(* Logix 5000 project; controller AMANA_DC_PLANT_01 vendor 1 type 14 code 164 rev 31.12; software revision 31.02; part 5 of 9 *)
(* tags used below, declared in another part *)
   Break_1stStation : BOOL;
   LN00_to_DC1_Main_Messages_5 : DINT[120];
   LN00_to_DC1_Main_Messages_6 : DINT[120];
   LN00DEM06 : DINT;
   LN00DEM07 : DINT;
   LN00DEM08 : DINT;
   LN00DEM09 : DINT;
   LN00DEM10 : DINT;
   LN00DEM11 : DINT;
   LN00DEM12 : DINT;
   LN00DEM13 : DINT;
   LN00DEM14 : DINT;
   LN00DEM15 : DINT;
   LN00DEM16 : DINT;
   LN00DEM17 : DINT;
   LN00DEM18 : DINT;
   LN00DEM19 : DINT;
   LN00DEM20 : DINT;
   LN00DEM21 : DINT;
   LN00DEM22 : DINT;
   LN00DEM23 : DINT;
   LN00DEM24 : DINT;
   LN00DEM25 : DINT;
   LN00DEM26 : DINT;
   LN00DEM27 : DINT;
   LN00DEM28 : DINT;
   LN00DEM29 : DINT;
   LN00DEM30 : DINT;
   LN00DEM31 : DINT;
   LN00DEM32 : DINT;
   LN00DEM33 : DINT;
   LN00DEM34 : DINT;
   LN00DEM35 : DINT;
   LN00DEM36 : DINT;
   LN00DEM37 : DINT;
   LN00DEM38 : DINT;
   LN00DEM39 : DINT;
   LN00DEM40 : DINT;
   LN00DEM41 : DINT;
   LN00DEM42 : DINT;
   LN00DEM43 : DINT;
   LN00DEM44 : DINT;
   LN00DEM45 : DINT;
   LN00DEM46 : DINT;
   LN00DEM47 : DINT;
   LN00DEM48 : DINT;
   LN00DEM49 : DINT;
   LN00DEM50 : DINT;
   LN00DEM51 : DINT;
   LN00DEM52 : DINT;
   LN00DEM53 : DINT;
   LN00DEM54 : DINT;
   LN00DEM55 : DINT;
   LN00DEM56 : DINT;
   LN00DEM57 : DINT;
   LN00DEM58 : DINT;
   LN00DEM59 : DINT;
   LN00DEM60 : DINT;
   LN00DEM61 : DINT;
   LN00DEM62 : DINT;
   LN00DEM63 : DINT;
   LN00DEM64 : DINT;
   LN00DEM65 : DINT;
   LN00DEM66 : DINT;
   LN00DEM67 : DINT;
   LN00DEM68 : DINT;
   LN00DEM69 : DINT;
   LN00DEM70 : DINT;
   LN00DEM71 : DINT;
   LN00DEM72 : DINT;
   LN00DEM73 : DINT;
   LN00DEM74 : DINT;
   LN00DEM75 : DINT;
   LN00DEM76 : DINT;
   LN00DEM77 : DINT;
   LN00DEM78 : DINT;
   LN00DEM79 : DINT;
   LN00DEM80 : DINT;
   LN00DEM81 : DINT;
   LN00DEM82 : DINT;
   LN00DEM83 : DINT;
   LN00DEM84 : DINT;
   LN00DEM85 : DINT;
   LN00DEM86 : DINT;
   LN00DEM87 : DINT;
   LN00DEM88 : DINT;
   LN00DEM89 : DINT;
   LN00DEM90 : DINT;
   LN00DEM91 : DINT;
   LN00DEM92 : DINT;
   LN00DEM93 : DINT;
   LN00DEM94 : DINT;
   LN00DEM95 : DINT;
   LN00DEM96 : DINT;
   LN00DEM97 : DINT;
   LN00DEM98 : DINT;
   LN00DFM01 : DINT;
   LN00DFM02 : DINT;
   LN00DFM03 : DINT;
(* LN00, continued *)

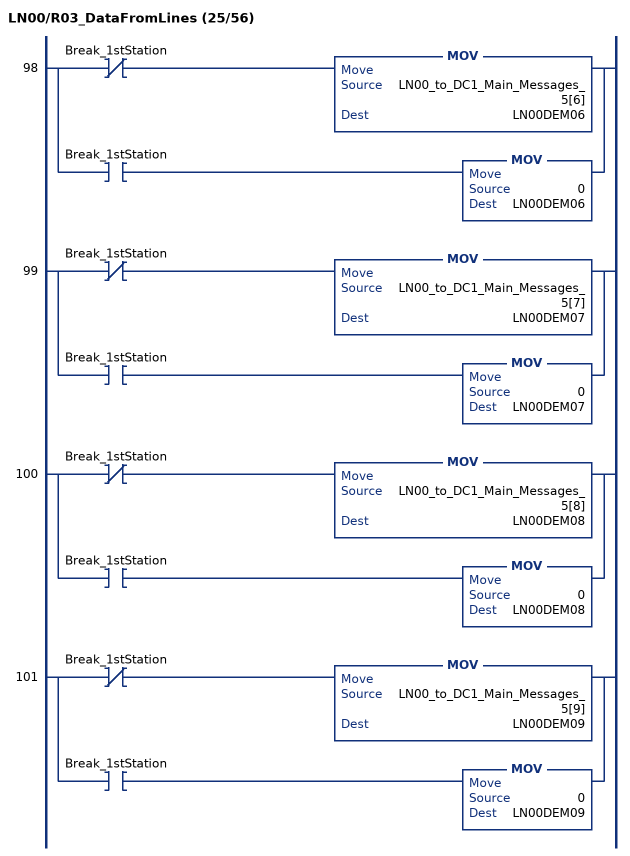
   [picture p71: LN00/R03_DataFromLines rungs 98-101]
   98: [XIO(Break_1stStation) MOV(LN00_to_DC1_Main_Messages_5[6],LN00DEM06) ,XIC(Break_1stStation) MOV(0,LN00DEM06) ];
   99: [XIO(Break_1stStation) MOV(LN00_to_DC1_Main_Messages_5[7],LN00DEM07) ,XIC(Break_1stStation) MOV(0,LN00DEM07) ];
   100: [XIO(Break_1stStation) MOV(LN00_to_DC1_Main_Messages_5[8],LN00DEM08) ,XIC(Break_1stStation) MOV(0,LN00DEM08) ];
   101: [XIO(Break_1stStation) MOV(LN00_to_DC1_Main_Messages_5[9],LN00DEM09) ,XIC(Break_1stStation) MOV(0,LN00DEM09) ];
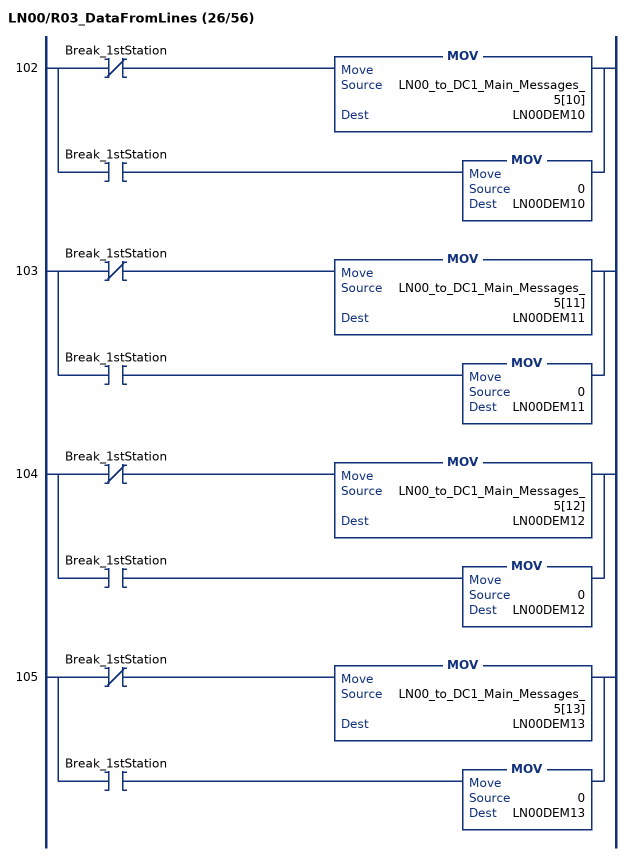
   102: [XIO(Break_1stStation) MOV(LN00_to_DC1_Main_Messages_5[10],LN00DEM10) ,XIC(Break_1stStation) MOV(0,LN00DEM10) ];
   103: [XIO(Break_1stStation) MOV(LN00_to_DC1_Main_Messages_5[11],LN00DEM11) ,XIC(Break_1stStation) MOV(0,LN00DEM11) ];
   104: [XIO(Break_1stStation) MOV(LN00_to_DC1_Main_Messages_5[12],LN00DEM12) ,XIC(Break_1stStation) MOV(0,LN00DEM12) ];
   105: [XIO(Break_1stStation) MOV(LN00_to_DC1_Main_Messages_5[13],LN00DEM13) ,XIC(Break_1stStation) MOV(0,LN00DEM13) ];
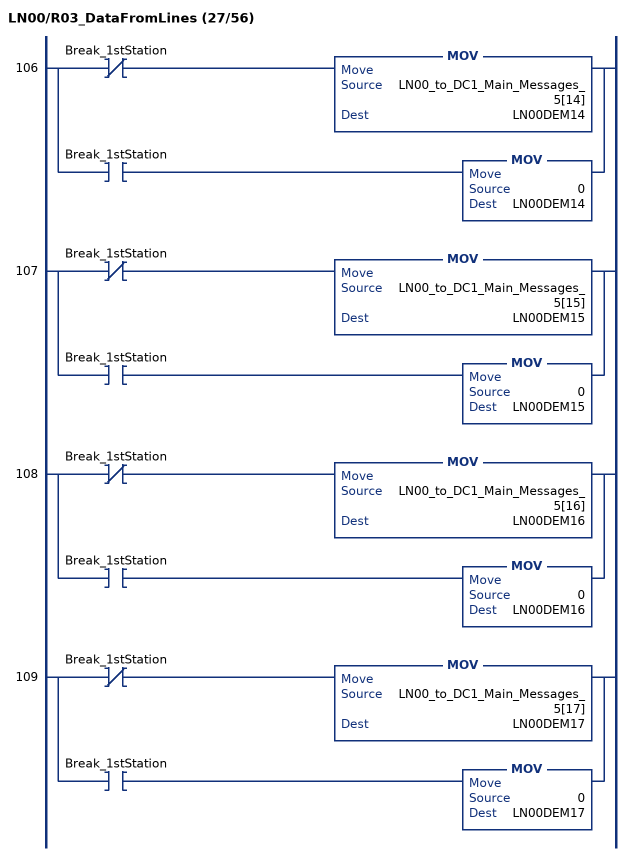
   106: [XIO(Break_1stStation) MOV(LN00_to_DC1_Main_Messages_5[14],LN00DEM14) ,XIC(Break_1stStation) MOV(0,LN00DEM14) ];
   107: [XIO(Break_1stStation) MOV(LN00_to_DC1_Main_Messages_5[15],LN00DEM15) ,XIC(Break_1stStation) MOV(0,LN00DEM15) ];
   108: [XIO(Break_1stStation) MOV(LN00_to_DC1_Main_Messages_5[16],LN00DEM16) ,XIC(Break_1stStation) MOV(0,LN00DEM16) ];
   109: [XIO(Break_1stStation) MOV(LN00_to_DC1_Main_Messages_5[17],LN00DEM17) ,XIC(Break_1stStation) MOV(0,LN00DEM17) ];
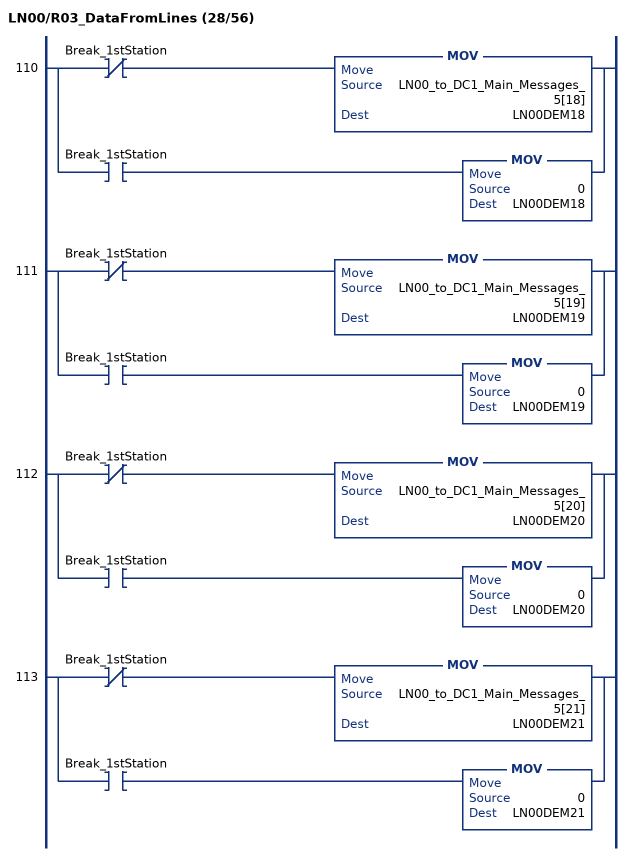
   110: [XIO(Break_1stStation) MOV(LN00_to_DC1_Main_Messages_5[18],LN00DEM18) ,XIC(Break_1stStation) MOV(0,LN00DEM18) ];
   111: [XIO(Break_1stStation) MOV(LN00_to_DC1_Main_Messages_5[19],LN00DEM19) ,XIC(Break_1stStation) MOV(0,LN00DEM19) ];
   112: [XIO(Break_1stStation) MOV(LN00_to_DC1_Main_Messages_5[20],LN00DEM20) ,XIC(Break_1stStation) MOV(0,LN00DEM20) ];
   113: [XIO(Break_1stStation) MOV(LN00_to_DC1_Main_Messages_5[21],LN00DEM21) ,XIC(Break_1stStation) MOV(0,LN00DEM21) ];
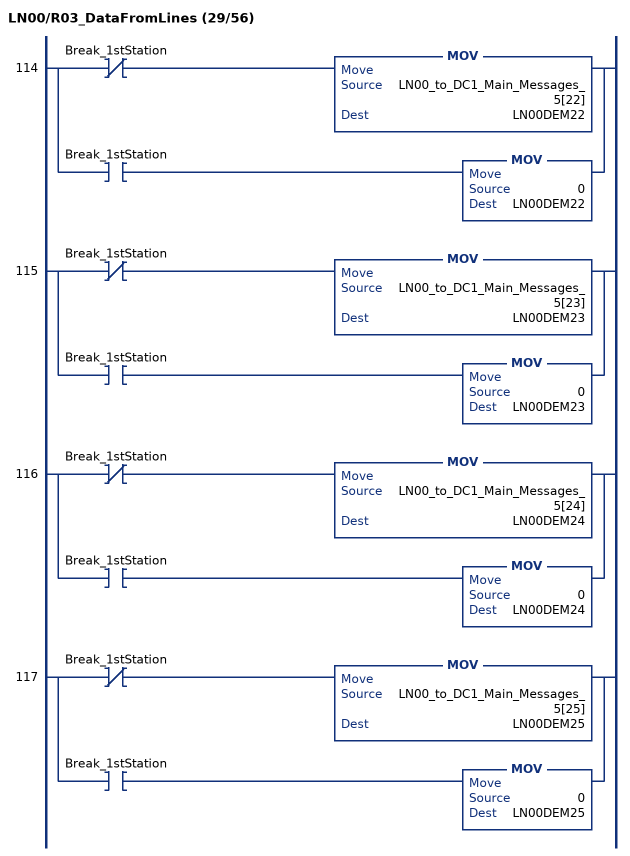
   114: [XIO(Break_1stStation) MOV(LN00_to_DC1_Main_Messages_5[22],LN00DEM22) ,XIC(Break_1stStation) MOV(0,LN00DEM22) ];
   115: [XIO(Break_1stStation) MOV(LN00_to_DC1_Main_Messages_5[23],LN00DEM23) ,XIC(Break_1stStation) MOV(0,LN00DEM23) ];
   116: [XIO(Break_1stStation) MOV(LN00_to_DC1_Main_Messages_5[24],LN00DEM24) ,XIC(Break_1stStation) MOV(0,LN00DEM24) ];
   117: [XIO(Break_1stStation) MOV(LN00_to_DC1_Main_Messages_5[25],LN00DEM25) ,XIC(Break_1stStation) MOV(0,LN00DEM25) ];
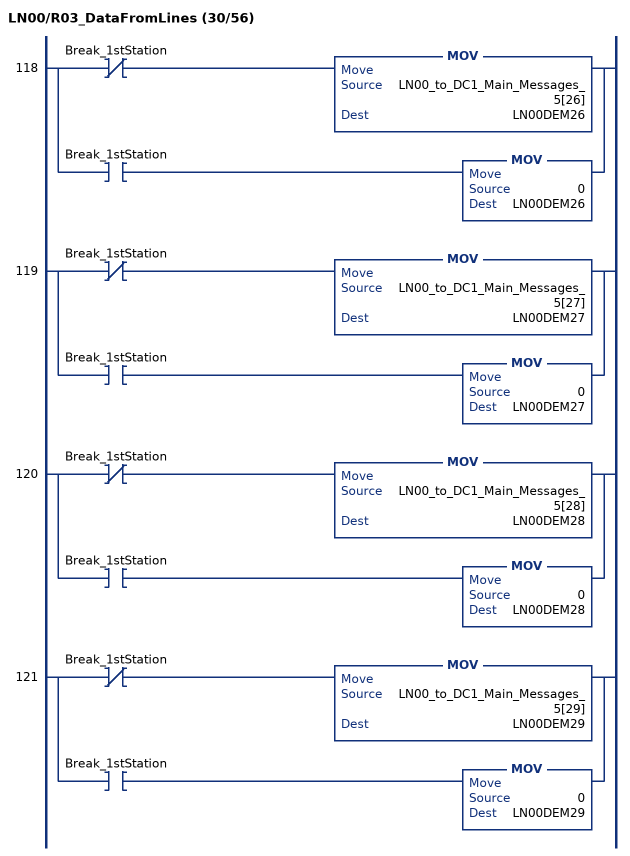
   118: [XIO(Break_1stStation) MOV(LN00_to_DC1_Main_Messages_5[26],LN00DEM26) ,XIC(Break_1stStation) MOV(0,LN00DEM26) ];
   119: [XIO(Break_1stStation) MOV(LN00_to_DC1_Main_Messages_5[27],LN00DEM27) ,XIC(Break_1stStation) MOV(0,LN00DEM27) ];
   120: [XIO(Break_1stStation) MOV(LN00_to_DC1_Main_Messages_5[28],LN00DEM28) ,XIC(Break_1stStation) MOV(0,LN00DEM28) ];
   121: [XIO(Break_1stStation) MOV(LN00_to_DC1_Main_Messages_5[29],LN00DEM29) ,XIC(Break_1stStation) MOV(0,LN00DEM29) ];
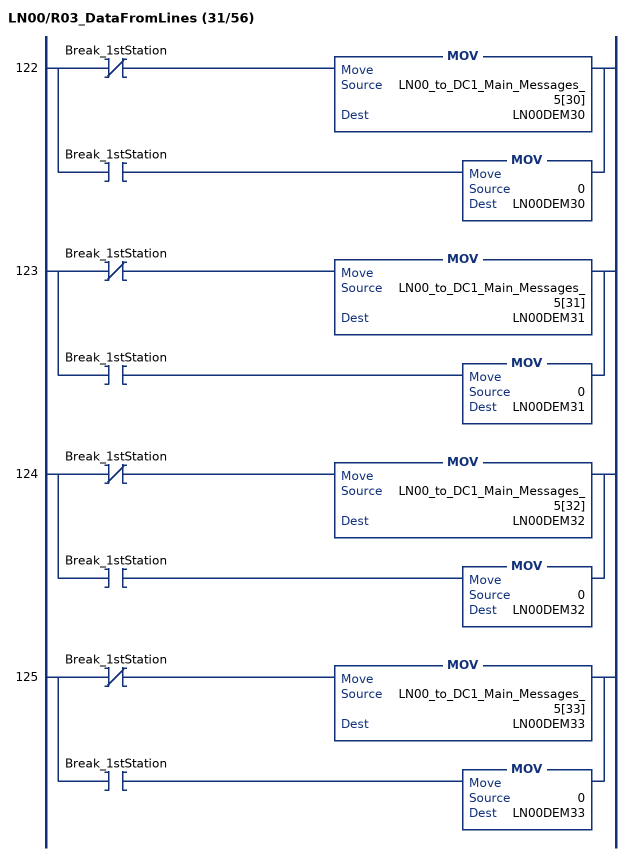
   122: [XIO(Break_1stStation) MOV(LN00_to_DC1_Main_Messages_5[30],LN00DEM30) ,XIC(Break_1stStation) MOV(0,LN00DEM30) ];
   123: [XIO(Break_1stStation) MOV(LN00_to_DC1_Main_Messages_5[31],LN00DEM31) ,XIC(Break_1stStation) MOV(0,LN00DEM31) ];
   124: [XIO(Break_1stStation) MOV(LN00_to_DC1_Main_Messages_5[32],LN00DEM32) ,XIC(Break_1stStation) MOV(0,LN00DEM32) ];
   125: [XIO(Break_1stStation) MOV(LN00_to_DC1_Main_Messages_5[33],LN00DEM33) ,XIC(Break_1stStation) MOV(0,LN00DEM33) ];
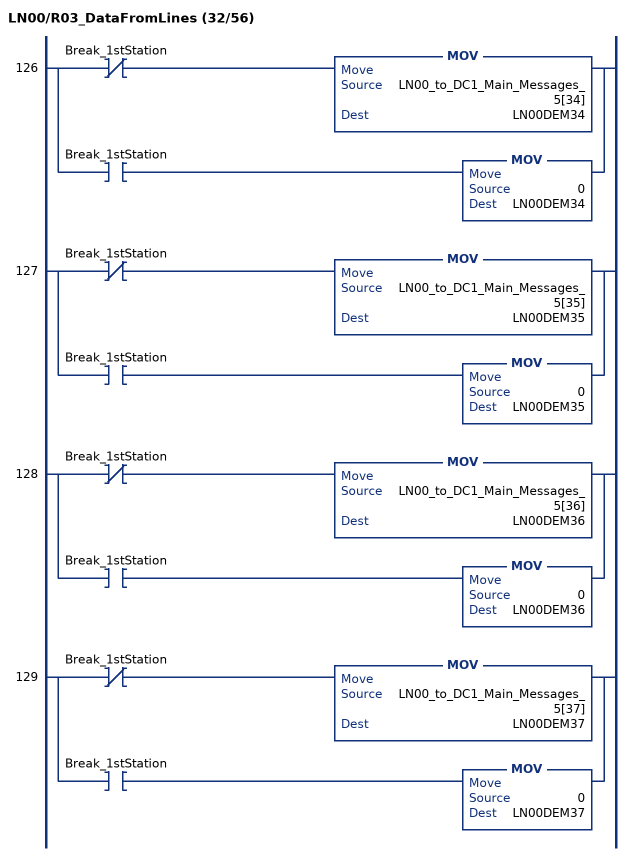
   126: [XIO(Break_1stStation) MOV(LN00_to_DC1_Main_Messages_5[34],LN00DEM34) ,XIC(Break_1stStation) MOV(0,LN00DEM34) ];
   127: [XIO(Break_1stStation) MOV(LN00_to_DC1_Main_Messages_5[35],LN00DEM35) ,XIC(Break_1stStation) MOV(0,LN00DEM35) ];
   128: [XIO(Break_1stStation) MOV(LN00_to_DC1_Main_Messages_5[36],LN00DEM36) ,XIC(Break_1stStation) MOV(0,LN00DEM36) ];
   129: [XIO(Break_1stStation) MOV(LN00_to_DC1_Main_Messages_5[37],LN00DEM37) ,XIC(Break_1stStation) MOV(0,LN00DEM37) ];
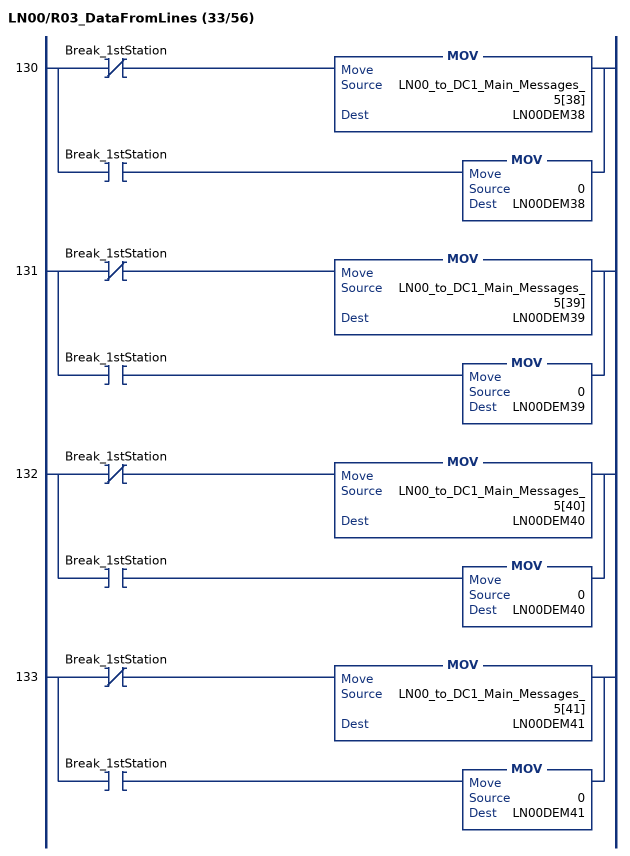
   130: [XIO(Break_1stStation) MOV(LN00_to_DC1_Main_Messages_5[38],LN00DEM38) ,XIC(Break_1stStation) MOV(0,LN00DEM38) ];
   131: [XIO(Break_1stStation) MOV(LN00_to_DC1_Main_Messages_5[39],LN00DEM39) ,XIC(Break_1stStation) MOV(0,LN00DEM39) ];
   132: [XIO(Break_1stStation) MOV(LN00_to_DC1_Main_Messages_5[40],LN00DEM40) ,XIC(Break_1stStation) MOV(0,LN00DEM40) ];
   133: [XIO(Break_1stStation) MOV(LN00_to_DC1_Main_Messages_5[41],LN00DEM41) ,XIC(Break_1stStation) MOV(0,LN00DEM41) ];
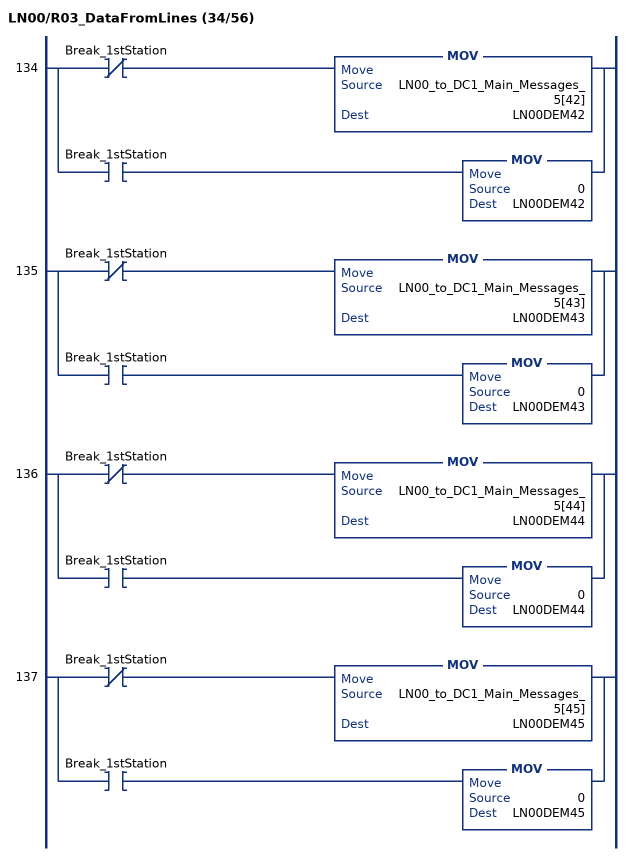
   134: [XIO(Break_1stStation) MOV(LN00_to_DC1_Main_Messages_5[42],LN00DEM42) ,XIC(Break_1stStation) MOV(0,LN00DEM42) ];
   135: [XIO(Break_1stStation) MOV(LN00_to_DC1_Main_Messages_5[43],LN00DEM43) ,XIC(Break_1stStation) MOV(0,LN00DEM43) ];
   136: [XIO(Break_1stStation) MOV(LN00_to_DC1_Main_Messages_5[44],LN00DEM44) ,XIC(Break_1stStation) MOV(0,LN00DEM44) ];
   137: [XIO(Break_1stStation) MOV(LN00_to_DC1_Main_Messages_5[45],LN00DEM45) ,XIC(Break_1stStation) MOV(0,LN00DEM45) ];
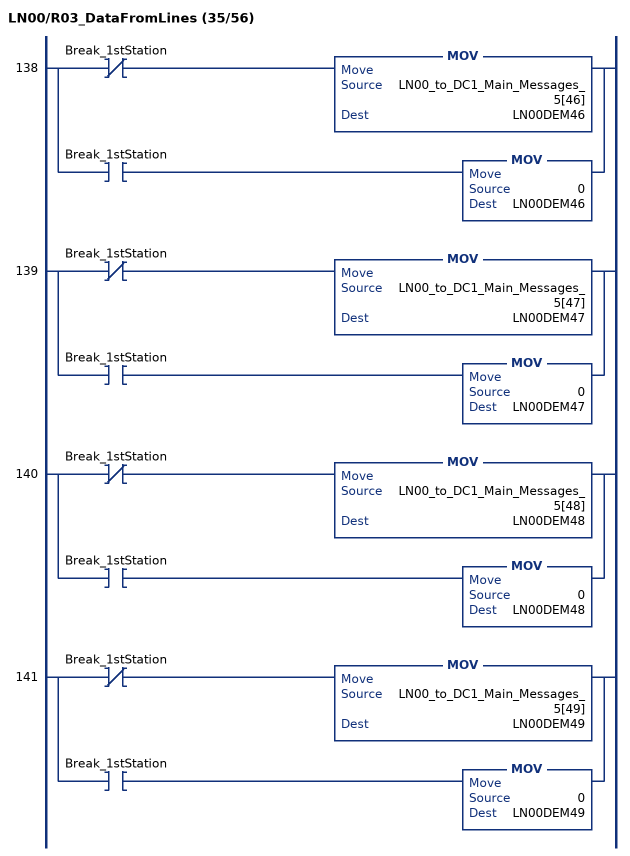
   138: [XIO(Break_1stStation) MOV(LN00_to_DC1_Main_Messages_5[46],LN00DEM46) ,XIC(Break_1stStation) MOV(0,LN00DEM46) ];
   139: [XIO(Break_1stStation) MOV(LN00_to_DC1_Main_Messages_5[47],LN00DEM47) ,XIC(Break_1stStation) MOV(0,LN00DEM47) ];
   140: [XIO(Break_1stStation) MOV(LN00_to_DC1_Main_Messages_5[48],LN00DEM48) ,XIC(Break_1stStation) MOV(0,LN00DEM48) ];
   141: [XIO(Break_1stStation) MOV(LN00_to_DC1_Main_Messages_5[49],LN00DEM49) ,XIC(Break_1stStation) MOV(0,LN00DEM49) ];
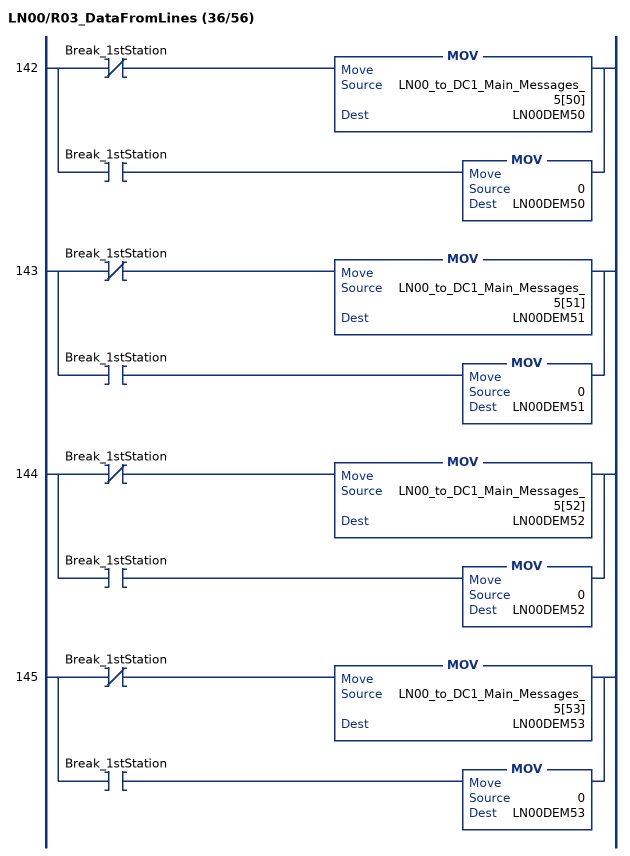
   142: [XIO(Break_1stStation) MOV(LN00_to_DC1_Main_Messages_5[50],LN00DEM50) ,XIC(Break_1stStation) MOV(0,LN00DEM50) ];
   143: [XIO(Break_1stStation) MOV(LN00_to_DC1_Main_Messages_5[51],LN00DEM51) ,XIC(Break_1stStation) MOV(0,LN00DEM51) ];
   144: [XIO(Break_1stStation) MOV(LN00_to_DC1_Main_Messages_5[52],LN00DEM52) ,XIC(Break_1stStation) MOV(0,LN00DEM52) ];
   145: [XIO(Break_1stStation) MOV(LN00_to_DC1_Main_Messages_5[53],LN00DEM53) ,XIC(Break_1stStation) MOV(0,LN00DEM53) ];
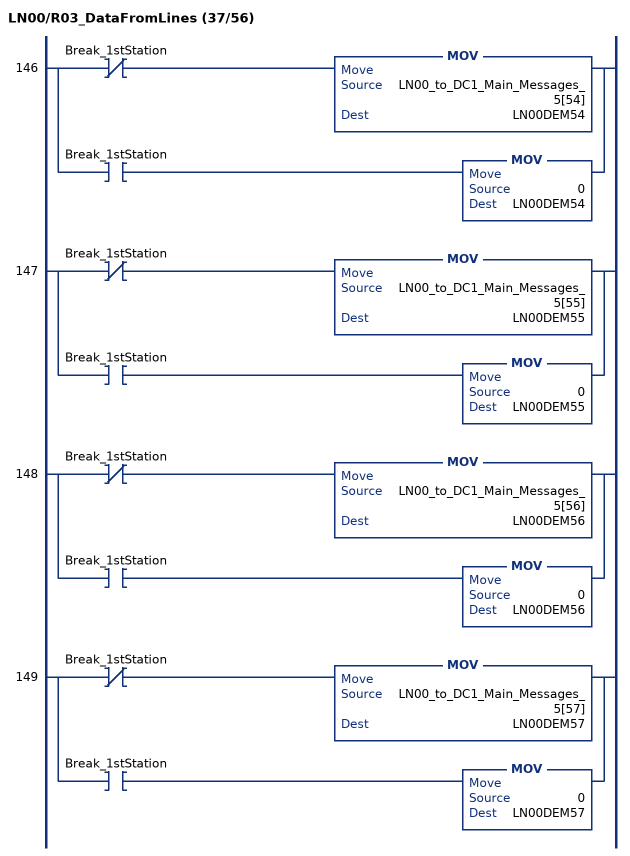
   146: [XIO(Break_1stStation) MOV(LN00_to_DC1_Main_Messages_5[54],LN00DEM54) ,XIC(Break_1stStation) MOV(0,LN00DEM54) ];
   147: [XIO(Break_1stStation) MOV(LN00_to_DC1_Main_Messages_5[55],LN00DEM55) ,XIC(Break_1stStation) MOV(0,LN00DEM55) ];
   148: [XIO(Break_1stStation) MOV(LN00_to_DC1_Main_Messages_5[56],LN00DEM56) ,XIC(Break_1stStation) MOV(0,LN00DEM56) ];
   149: [XIO(Break_1stStation) MOV(LN00_to_DC1_Main_Messages_5[57],LN00DEM57) ,XIC(Break_1stStation) MOV(0,LN00DEM57) ];
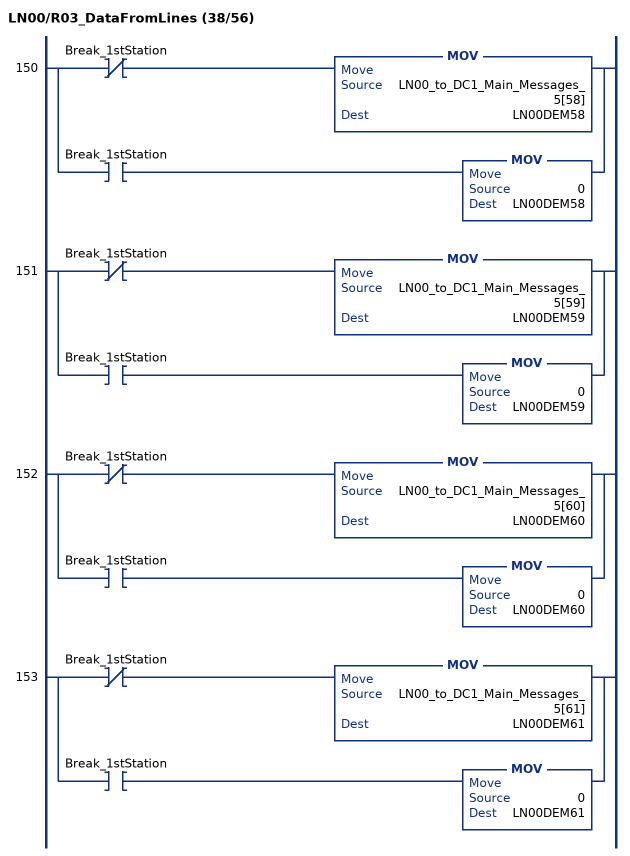
   150: [XIO(Break_1stStation) MOV(LN00_to_DC1_Main_Messages_5[58],LN00DEM58) ,XIC(Break_1stStation) MOV(0,LN00DEM58) ];
   151: [XIO(Break_1stStation) MOV(LN00_to_DC1_Main_Messages_5[59],LN00DEM59) ,XIC(Break_1stStation) MOV(0,LN00DEM59) ];
   152: [XIO(Break_1stStation) MOV(LN00_to_DC1_Main_Messages_5[60],LN00DEM60) ,XIC(Break_1stStation) MOV(0,LN00DEM60) ];
   153: [XIO(Break_1stStation) MOV(LN00_to_DC1_Main_Messages_5[61],LN00DEM61) ,XIC(Break_1stStation) MOV(0,LN00DEM61) ];
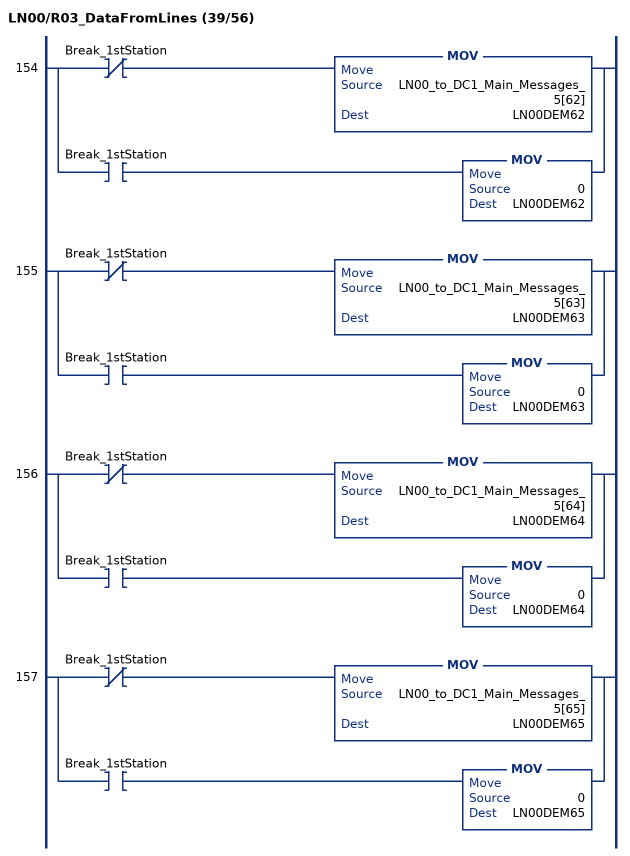
   154: [XIO(Break_1stStation) MOV(LN00_to_DC1_Main_Messages_5[62],LN00DEM62) ,XIC(Break_1stStation) MOV(0,LN00DEM62) ];
   155: [XIO(Break_1stStation) MOV(LN00_to_DC1_Main_Messages_5[63],LN00DEM63) ,XIC(Break_1stStation) MOV(0,LN00DEM63) ];
   156: [XIO(Break_1stStation) MOV(LN00_to_DC1_Main_Messages_5[64],LN00DEM64) ,XIC(Break_1stStation) MOV(0,LN00DEM64) ];
   157: [XIO(Break_1stStation) MOV(LN00_to_DC1_Main_Messages_5[65],LN00DEM65) ,XIC(Break_1stStation) MOV(0,LN00DEM65) ];
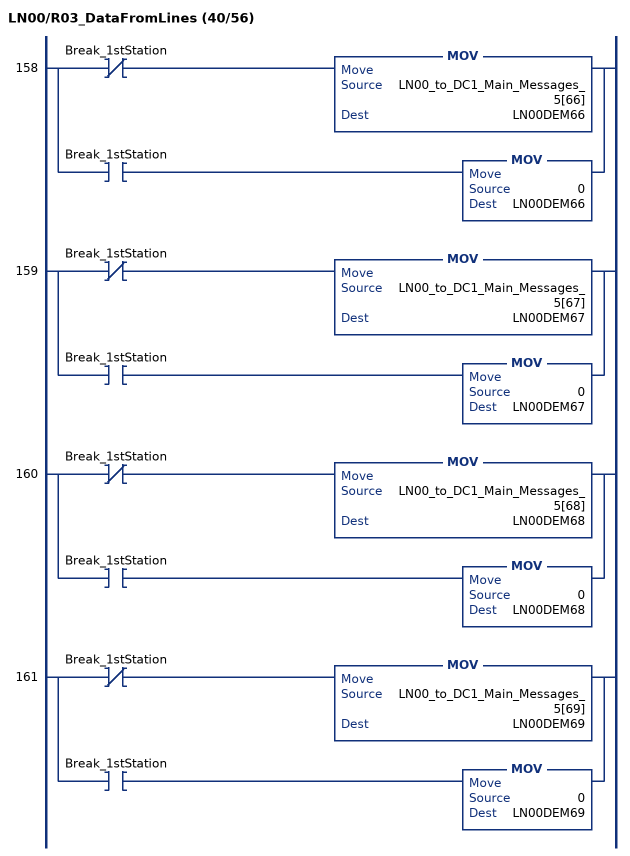
   158: [XIO(Break_1stStation) MOV(LN00_to_DC1_Main_Messages_5[66],LN00DEM66) ,XIC(Break_1stStation) MOV(0,LN00DEM66) ];
   159: [XIO(Break_1stStation) MOV(LN00_to_DC1_Main_Messages_5[67],LN00DEM67) ,XIC(Break_1stStation) MOV(0,LN00DEM67) ];
   160: [XIO(Break_1stStation) MOV(LN00_to_DC1_Main_Messages_5[68],LN00DEM68) ,XIC(Break_1stStation) MOV(0,LN00DEM68) ];
   161: [XIO(Break_1stStation) MOV(LN00_to_DC1_Main_Messages_5[69],LN00DEM69) ,XIC(Break_1stStation) MOV(0,LN00DEM69) ];
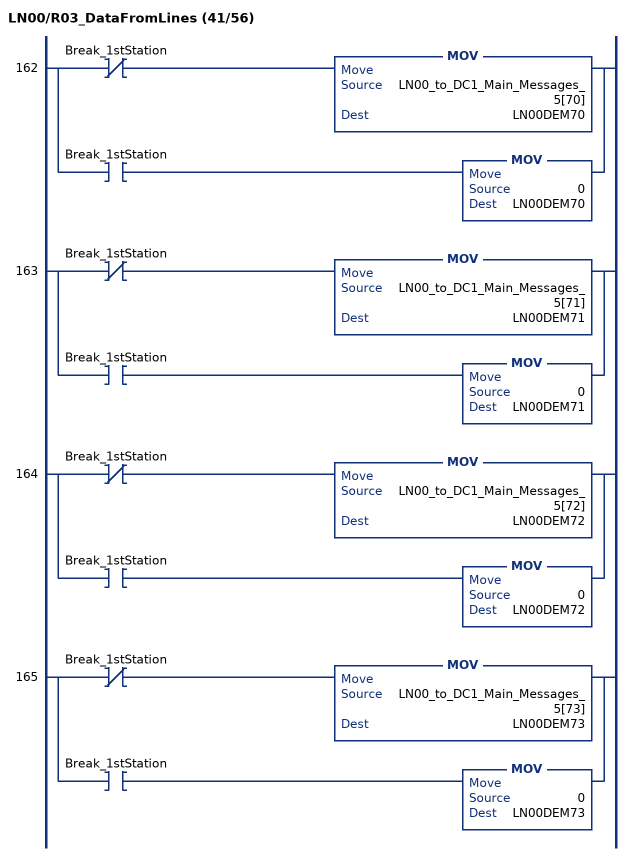
   162: [XIO(Break_1stStation) MOV(LN00_to_DC1_Main_Messages_5[70],LN00DEM70) ,XIC(Break_1stStation) MOV(0,LN00DEM70) ];
   163: [XIO(Break_1stStation) MOV(LN00_to_DC1_Main_Messages_5[71],LN00DEM71) ,XIC(Break_1stStation) MOV(0,LN00DEM71) ];
   164: [XIO(Break_1stStation) MOV(LN00_to_DC1_Main_Messages_5[72],LN00DEM72) ,XIC(Break_1stStation) MOV(0,LN00DEM72) ];
   165: [XIO(Break_1stStation) MOV(LN00_to_DC1_Main_Messages_5[73],LN00DEM73) ,XIC(Break_1stStation) MOV(0,LN00DEM73) ];
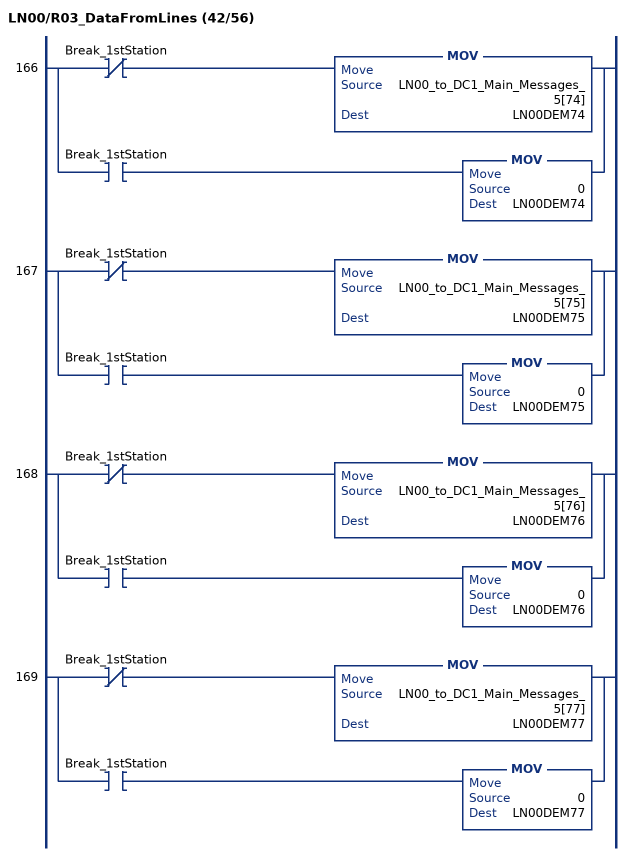
   166: [XIO(Break_1stStation) MOV(LN00_to_DC1_Main_Messages_5[74],LN00DEM74) ,XIC(Break_1stStation) MOV(0,LN00DEM74) ];
   167: [XIO(Break_1stStation) MOV(LN00_to_DC1_Main_Messages_5[75],LN00DEM75) ,XIC(Break_1stStation) MOV(0,LN00DEM75) ];
   168: [XIO(Break_1stStation) MOV(LN00_to_DC1_Main_Messages_5[76],LN00DEM76) ,XIC(Break_1stStation) MOV(0,LN00DEM76) ];
   169: [XIO(Break_1stStation) MOV(LN00_to_DC1_Main_Messages_5[77],LN00DEM77) ,XIC(Break_1stStation) MOV(0,LN00DEM77) ];
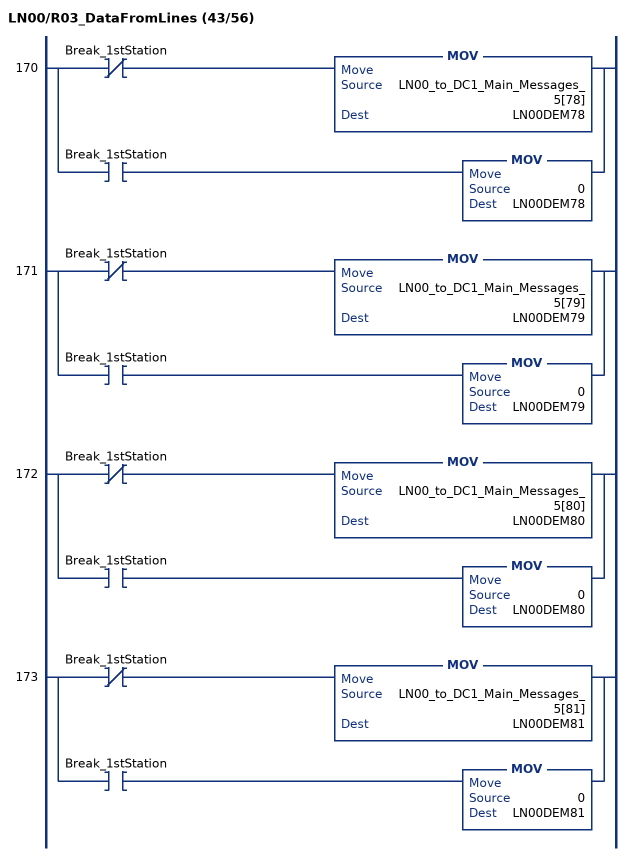
   170: [XIO(Break_1stStation) MOV(LN00_to_DC1_Main_Messages_5[78],LN00DEM78) ,XIC(Break_1stStation) MOV(0,LN00DEM78) ];
   171: [XIO(Break_1stStation) MOV(LN00_to_DC1_Main_Messages_5[79],LN00DEM79) ,XIC(Break_1stStation) MOV(0,LN00DEM79) ];
   172: [XIO(Break_1stStation) MOV(LN00_to_DC1_Main_Messages_5[80],LN00DEM80) ,XIC(Break_1stStation) MOV(0,LN00DEM80) ];
   173: [XIO(Break_1stStation) MOV(LN00_to_DC1_Main_Messages_5[81],LN00DEM81) ,XIC(Break_1stStation) MOV(0,LN00DEM81) ];
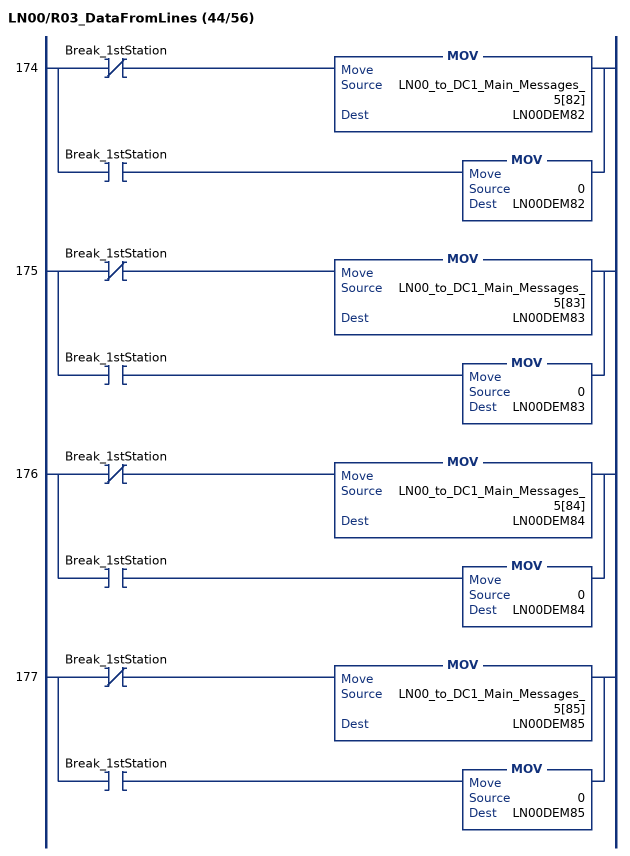
   174: [XIO(Break_1stStation) MOV(LN00_to_DC1_Main_Messages_5[82],LN00DEM82) ,XIC(Break_1stStation) MOV(0,LN00DEM82) ];
   175: [XIO(Break_1stStation) MOV(LN00_to_DC1_Main_Messages_5[83],LN00DEM83) ,XIC(Break_1stStation) MOV(0,LN00DEM83) ];
   176: [XIO(Break_1stStation) MOV(LN00_to_DC1_Main_Messages_5[84],LN00DEM84) ,XIC(Break_1stStation) MOV(0,LN00DEM84) ];
   177: [XIO(Break_1stStation) MOV(LN00_to_DC1_Main_Messages_5[85],LN00DEM85) ,XIC(Break_1stStation) MOV(0,LN00DEM85) ];
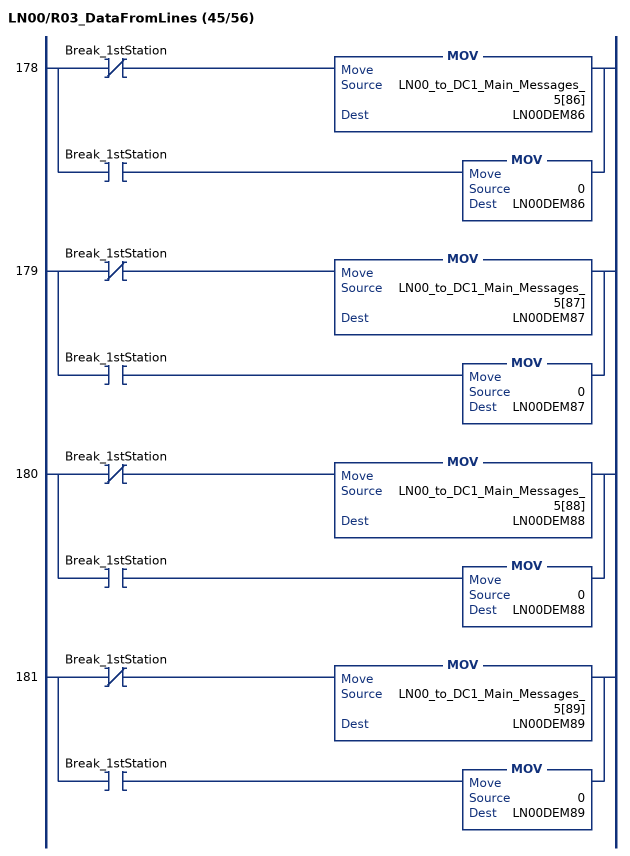
   178: [XIO(Break_1stStation) MOV(LN00_to_DC1_Main_Messages_5[86],LN00DEM86) ,XIC(Break_1stStation) MOV(0,LN00DEM86) ];
   179: [XIO(Break_1stStation) MOV(LN00_to_DC1_Main_Messages_5[87],LN00DEM87) ,XIC(Break_1stStation) MOV(0,LN00DEM87) ];
   180: [XIO(Break_1stStation) MOV(LN00_to_DC1_Main_Messages_5[88],LN00DEM88) ,XIC(Break_1stStation) MOV(0,LN00DEM88) ];
   181: [XIO(Break_1stStation) MOV(LN00_to_DC1_Main_Messages_5[89],LN00DEM89) ,XIC(Break_1stStation) MOV(0,LN00DEM89) ];
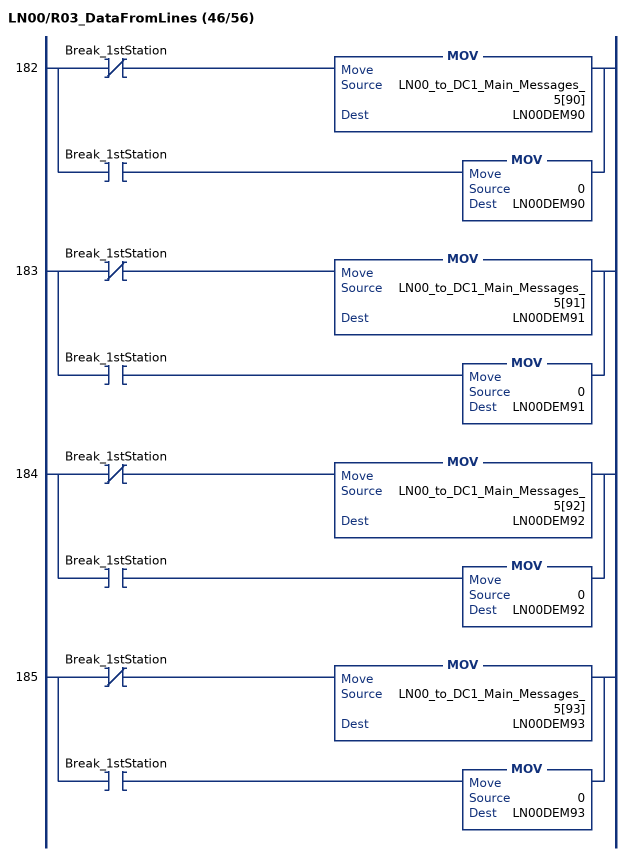
   182: [XIO(Break_1stStation) MOV(LN00_to_DC1_Main_Messages_5[90],LN00DEM90) ,XIC(Break_1stStation) MOV(0,LN00DEM90) ];
   183: [XIO(Break_1stStation) MOV(LN00_to_DC1_Main_Messages_5[91],LN00DEM91) ,XIC(Break_1stStation) MOV(0,LN00DEM91) ];
   184: [XIO(Break_1stStation) MOV(LN00_to_DC1_Main_Messages_5[92],LN00DEM92) ,XIC(Break_1stStation) MOV(0,LN00DEM92) ];
   185: [XIO(Break_1stStation) MOV(LN00_to_DC1_Main_Messages_5[93],LN00DEM93) ,XIC(Break_1stStation) MOV(0,LN00DEM93) ];
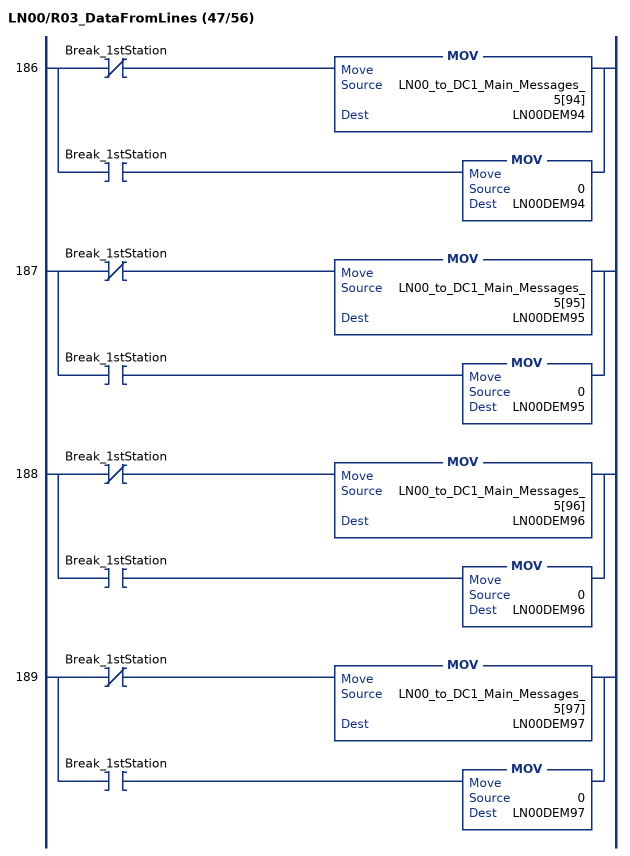
   186: [XIO(Break_1stStation) MOV(LN00_to_DC1_Main_Messages_5[94],LN00DEM94) ,XIC(Break_1stStation) MOV(0,LN00DEM94) ];
   187: [XIO(Break_1stStation) MOV(LN00_to_DC1_Main_Messages_5[95],LN00DEM95) ,XIC(Break_1stStation) MOV(0,LN00DEM95) ];
   188: [XIO(Break_1stStation) MOV(LN00_to_DC1_Main_Messages_5[96],LN00DEM96) ,XIC(Break_1stStation) MOV(0,LN00DEM96) ];
   189: [XIO(Break_1stStation) MOV(LN00_to_DC1_Main_Messages_5[97],LN00DEM97) ,XIC(Break_1stStation) MOV(0,LN00DEM97) ];
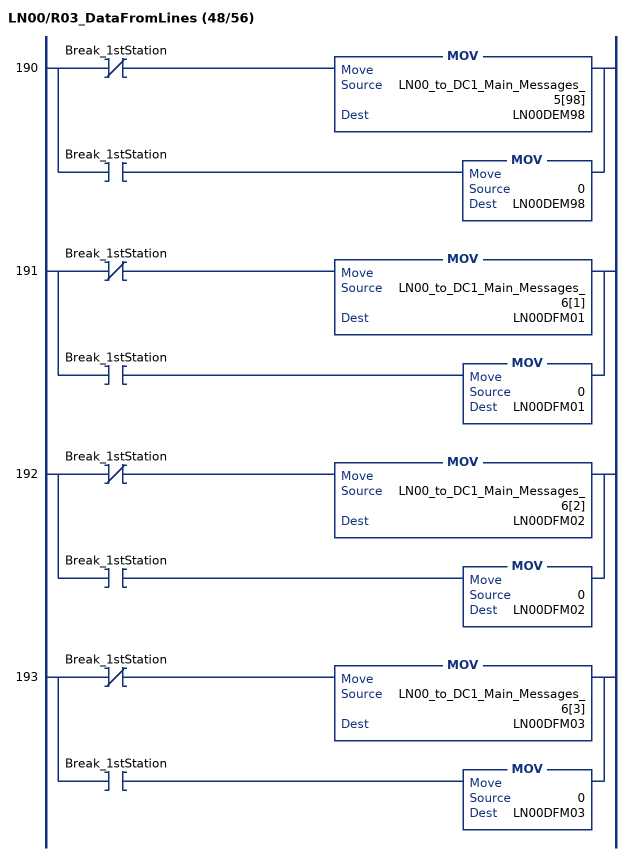
   190: [XIO(Break_1stStation) MOV(LN00_to_DC1_Main_Messages_5[98],LN00DEM98) ,XIC(Break_1stStation) MOV(0,LN00DEM98) ];
   191: [XIO(Break_1stStation) MOV(LN00_to_DC1_Main_Messages_6[1],LN00DFM01) ,XIC(Break_1stStation) MOV(0,LN00DFM01) ];
   192: [XIO(Break_1stStation) MOV(LN00_to_DC1_Main_Messages_6[2],LN00DFM02) ,XIC(Break_1stStation) MOV(0,LN00DFM02) ];
   193: [XIO(Break_1stStation) MOV(LN00_to_DC1_Main_Messages_6[3],LN00DFM03) ,XIC(Break_1stStation) MOV(0,LN00DFM03) ];
